FUNCTION_BLOCK T_MockBoolCommandTask IMPLEMENTS I_BoolResultTask
VAR_INPUT
  _Busy, _Done, _Error, _Timeout : BOOL;
  _Result : BOOL;
END_VAR

METHOD Abort
END_METHOD

PROPERTY Available : BOOL
GET
END_GET
END_PROPERTY

PROPERTY Busy : BOOL
GET
Busy := _busy;
END_GET
END_PROPERTY

METHOD CyclicLogic
END_METHOD

PROPERTY Done : BOOL
GET
Done := _Done;
END_GET
END_PROPERTY

PROPERTY Error : BOOL
GET
Error := _Error;
END_GET
END_PROPERTY

PROPERTY ErrorId : STRING
GET
END_GET
END_PROPERTY

METHOD Execute : BOOL
END_METHOD

METHOD Free
END_METHOD

PROPERTY Result : BOOL
GET
Result := _Result;
END_GET
END_PROPERTY

PROPERTY Timeout : BOOL
GET
Timeout := _Timeout;
END_GET
END_PROPERTY

END_FUNCTION_BLOCK

(* stored: Version 1.1.0.1
   POU T_MockBoolCommandTask: Id {efdcfd4f-1fbd-4bc6-aa24-a9c842552591}, SpecialFunc None
   Method Abort: Id {6adfd664-6386-4259-869f-b7d5e4babe43}
   Property Available: Id {57b0532b-5f22-47fb-bdbf-688f16e4d843}
   Get Get: Id {71e0aaa7-fa9d-4a62-8cb4-6637a3e4aa67}
   Property Busy: Id {20e149c3-7bda-4ede-a1aa-39088c8ed107}
   Get Get: Id {3f9f4856-f5fd-44bb-ae85-1b43734c47cb}
   Method CyclicLogic: Id {405a2a55-6734-4deb-bfd1-4d804017529e}
   Property Done: Id {902e8abc-4d44-44be-be10-f3cf4c058e8e}
   Get Get: Id {a64957e7-563b-4593-918e-f5853eba1a2a}
   Property Error: Id {3266b145-025e-4409-b119-fb2146efe6a8}
   Get Get: Id {43e48575-3fe6-444c-b8b2-6fba5917a6c8}
   Property ErrorId: Id {918f1f9b-3a41-4d2b-98e3-1bd3592008be}
   Get Get: Id {e794e974-384f-4df2-bd07-ad8ecc6d80e6}
   Method Execute: Id {697e00d6-98c3-4dfb-ba0d-74d8d71b5655}
   Method Free: Id {3724c141-e8a5-43b6-bf5f-a845567f8e3f}
   Property Result: Id {7685c52f-2572-4f2a-ad81-ffc9a6d411a9}
   Get Get: Id {0226efc7-ce3a-4afc-8f64-195a18c0be6b}
   Property Timeout: Id {94d72bfd-6de8-4221-bc87-2eb5996d16a8}
   Get Get: Id {fc4f3230-7de3-4c89-afd2-398f18d8c894} *)
